// TIA Portal V19 export
DATA_BLOCK "A0301_Trasporto"   // DB75
// stored: InstanceOfName A0301_Trasporto_FB, InstanceOfType FB
"A0301_Trasporto_FB"
   // VAR_INPUT
   //    AreaInterface : "AreaInterface";
   //    ZSI : "udt_ZoneSafetyInterface";
   //    DSI : "udt_DeviceSafetyInterface";
   //    Drive : "TAx_DriveInterface";
   //    DataIn : "SpeedMachine_DataIn";
   //    CIn : Struct
   //       Drive : "SpeedMachine_CIn";
   //       OP_SemiAut_PB : Bool;
   //    END_STRUCT;
   //    Config : "SpeedMachine_Config";
   //    HWID_Ax_TEL1 : HW_SUBMODULE;
   // END_VAR
   // VAR_OUTPUT
   //    MachineInterface { ExternalAccessible := 'False'; ExternalVisible := 'False'; ExternalWritable := 'False'} : "MachineInterface";
   //    COut : Struct
   //       Ax : "SpeedMachine_COut";
   //       Ax_VelOveride : Struct
   //          Enable : Bool;
   //          Value : Real;
   //       END_STRUCT;
   //    END_STRUCT;
   // END_VAR
   // VAR_IN_OUT
   //    Par : Struct
   //       Ax : "SpeedMachine_Par";
   //       Ax_Aut : "A0301_Mach_Speed_Par";
   //    END_STRUCT;
   // END_VAR
   // VAR
   //    Alarm : Struct
   //       Ax { ExternalVisible := 'False'} : "SpeedMachine_Alr";
   //    END_STRUCT;
   //    Warning : Struct
   //       Ax { S7_SetPoint := 'True'} : "SpeedMachine_Wng";
   //       OP_REST_MissingCnd : Bool;
   //       OP_WORK_MissingCnd : Bool;
   //    END_STRUCT;
   //    Ax : "SpeedMachine_FB";
   //    ValueVelOvr { ExternalAccessible := 'False'; ExternalVisible := 'False'; ExternalWritable := 'False'} : Array[1..10] of Real;
   //    Sts : Struct
   //       OP_CanMoveFreely : Bool;
   //       OP_Bwd_Cnd : Bool;
   //       OP_Fwd_Cnd : Bool;
   //    END_STRUCT;
   //    Ctrl : Struct
   //       OP_Bwd_Man : Bool;
   //       OP_Fwd_Man : Bool;
   //       OP_Bwd_Aut : Bool;
   //       OP_Fwd_Aut : Bool;
   //       OP_Bwd_Run : Bool;
   //       OP_Fwd_Run : Bool;
   //    END_STRUCT;
   //    AUX : Struct
   //       OP_Bwd_PB : Bool;
   //       OP_Fwd_PB : Bool;
   //    END_STRUCT;
   //    TON_OP_REST_MissingCnd { S7_SetPoint := 'True'} : TON_TIME;
   //    TON_OP_WORK_MissingCnd { S7_SetPoint := 'True'} : TON_TIME;
   // END_VAR
BEGIN
END_DATA_BLOCK
